FUNCTION F_Temp_Write_Value : ST_Modbus_Send_Frame
VAR_INPUT
	Module_Number	:BYTE;
	Command_Index	:WORD;
	Write_Value		:WORD;
END_VAR
VAR
END_VAR

F_Temp_Write_Value.UnitID	:= Module_Number;
F_Temp_Write_Value.StartAddress	:= Command_Index;
F_Temp_Write_Value.sendQuantity	:= 1;
F_Temp_Write_Value.SendData[0]	:= Write_Value;

END_FUNCTION

(* stored: Version 1.1.0.1
   POU F_Temp_Write_Value: Id {6edb265b-ff92-40fc-8087-9a6bc2b62562}, SpecialFunc None *)
